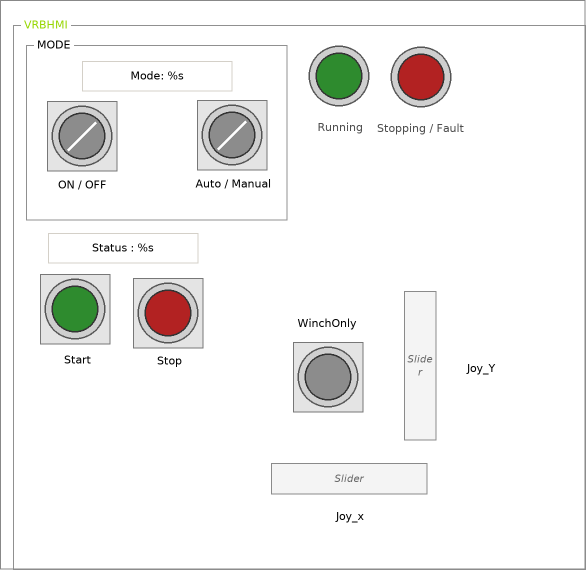
VISUALIZATION VirtualBoxHMI  // 586x570
    GroupBox (13,17 573x553), "VRBHMI"
        PushSwitch (27,257 70x70), variable: HMI.stVisuParam.bStart, behaviour: TAP, style: Switch-PushSwitch-Green
        PushSwitch (120,261 70x70), variable: HMI.stVisuParam.bStop, behaviour: TAP, style: Switch-PushSwitch-Red
        Lamp1 (291,24 70x70), variable: HMI.stVisuParam.bRunning, style: Lamp-Lamp1-Green
        Lamp1 (373,25 70x70), variable: HMI.stVisuParam.bStop, style: Lamp-Lamp1-Red
        Slider (5682,5127 161x29), scale 0..100
        Slider (5815,4955 30x143), scale 0..100
        Label (5690,5182 150x30), "Joy_X"
        Label (5852,4969 65x118), "Joy_Y"
        Label (360,97 95x29), "Stopping / Fault"
        Label (105,330 103x28), "Stop"
        Label (19,328 91x30), "Start"
        GroupBox (13,20 261x183), "MODE"
            Label (11,133 91x30), "ON / OFF"
            RotarySwitch (171,63 70x70), variable: HMI.stVisuParam.bAuto, behaviour: TOGGLE, style: Switch-RotarySwitch-Gray
            Label (162,132 91x30), "Auto / Manual"
            Textfield (56,24 150x30), "Mode: %s", text variable: HMI.eMode
            RotarySwitch (21,64 70x70), variable: HMI.stVisuParam.bOn, behaviour: TOGGLE, style: Switch-RotarySwitch-Gray
        Textfield (35,216 150x30), "Status : %s", text variable: HMI.eStatus
        Label (193,329 103x28)
        Label (280,96 95x29), "Running"
        Slider (258,446 156x31), variable: HMI.stVisuParam.fJoy_X, scale -1..1
        Slider (391,274 32x149), variable: HMI.stVisuParam.fJoy_Y, scale -1..1
        Label (298,484 78x31), "Joy_x"
        Label (433,338 70x27), "Joy_Y"
        PushSwitch (280,325 70x70), variable: HMI.stVisuParam.bTopSwitchJoy, behaviour: TOGGLE, style: Switch-PushSwitch-Gray
        Label (279,293 70x27), "WinchOnly"
END_VISUALIZATION

(* stored: Version 1.1.0.1, ProductVersion 3.1.4024.12
   Visu VirtualBoxHMI: Id {86afc6a3-02e3-4d3b-b864-83f52426aa86} *)
